// TIA Portal V18 export
VAR_GLOBAL   // PLC tag table "06_RD-2"
   "iRD-2" AT %I1.3 : Bool;
   "oRD-2" AT %Q0.5 : Bool;
END_VAR
